Fanuc KAREL source: kt00453.KL

-- PROVISIONAL review KL for V940-1; original PC SHA256 afcf880b9487944d8d7b4a21e90edddb76416df4b69c8be5fa58b4911816ae9f
-- Incomplete behavior may be omitted. Consult companion uncertainty JSON. Do not deploy.
PROGRAM KT00453
%NOLOCKGROUP
VAR
  OUT : BOOLEAN
-- UNRESOLVED_DECL H1 type=002017
-- UNRESOLVED_DECL Y2 type=002018
BEGIN
  -- V9_ZERO_TABLE_METADATA_HINT layout=0001; no indexed target words; source/name/runtime held
  -- UNRESOLVED_PC offsets 5-19; opcodes 2E,22,9D,33,B4
  -- UNRESOLVED_PC offsets 24-38; opcodes 2E,22,9D,33,B2
  -- UNRESOLVED_PC offsets 43-68; opcodes 22,9D,33,B3,22,9D,33,B1,5C,23
  -- UNRESOLVED_PC offsets 73-77; opcodes 7F
END KT00453
